FUNCTION_BLOCK FB_AtomicNumberLookup_Test EXTENDS TcUnit.FB_TestSuite
VAR
END_VAR


GivenElementExpectCorrectAtomicNumber();


METHOD PRIVATE GivenElementExpectCorrectAtomicNumber
VAR
    nResult : INT;
END_VAR

TEST('GivenElementExpectCorrectAtomicNumber');

nResult := F_AtomicNumberLookup(
    sMaterialName := 'C'
);

AssertEquals_INT(
    Expected := 6,
    Actual := nResult,
    Message := 'Incorrect result.'
);

nResult := F_AtomicNumberLookup(
    sMaterialName := 'Cu'
);

AssertEquals_INT(
    Expected := 29,
    Actual := nResult,
    Message := 'Incorrect result.'
);

nResult := F_AtomicNumberLookup(
    sMaterialName := 'Be'
);

AssertEquals_INT(
    Expected := 4,
    Actual := nResult,
    Message := 'Incorrect result.'
);

TEST_FINISHED();
END_METHOD

END_FUNCTION_BLOCK

(* stored: Version 1.1.0.1
   POU FB_AtomicNumberLookup_Test: Id {db138c95-91dc-4ac9-8915-081c5b7d7b7f}, SpecialFunc None
   Method GivenElementExpectCorrectAtomicNumber: Id {a0ee5d0e-6518-499c-a879-48b83f6ffe3c} *)
